(* IEC 61131-3 sources: cybercode_codesys_lib/src/basic/signal, 4 files *)

(* ---- FB_NumericChangeDetector.st ---- *)
FUNCTION_BLOCK FB_NumericChangeDetector
VAR_INPUT
    irValue : REAL;          // Входное числовое значение для мониторинга
END_VAR
VAR_OUTPUT
    qxChangeDetected : BOOL; // Импульс при обнаружении изменения значения
END_VAR
VAR
    _rPreviousValue : REAL := 0.0;    // Предыдущее значение для сравнения
    _xFirstCycle : BOOL := TRUE;      // Флаг первого цикла выполнения
    _rt_Change : R_TRIG;              // Триггер для генерации импульса
    _xValueChanged : BOOL := FALSE;   // Внутренний флаг изменения
END_VAR

// Пропускаем первый цикл для корректной инициализации
IF _xFirstCycle THEN
    _rPreviousValue := irValue;
    _xFirstCycle := FALSE;
    _xValueChanged := FALSE;
ELSE
    // Проверяем изменение значения
    IF _rPreviousValue <> irValue THEN
        _xValueChanged := TRUE;
        _rPreviousValue := irValue;
    ELSE
        _xValueChanged := FALSE;
    END_IF
END_IF

// Генерируем импульс при изменении через R_TRIG
_rt_Change(CLK := _xValueChanged);
qxChangeDetected := _rt_Change.Q;

(* Получение текущего отслеживаемого значения *)
METHOD GetCurrentValue : REAL
VAR_INPUT
END_VAR
    GetCurrentValue := irValue;
END_METHOD

(* Получение предыдущего значения *)
METHOD GetPreviousValue : REAL
VAR_INPUT
END_VAR
    GetPreviousValue := _rPreviousValue;
END_METHOD

(* Получение разности между текущим и предыдущим значением *)
METHOD GetValueDifference : REAL
VAR_INPUT
END_VAR
    GetValueDifference := irValue - _rPreviousValue;
END_METHOD

(* Проверка увеличения значения *)
METHOD IsValueIncreased : BOOL
VAR_INPUT
END_VAR
    IsValueIncreased := _xValueChanged AND (irValue > _rPreviousValue);
END_METHOD

(* Проверка уменьшения значения *)
METHOD IsValueDecreased : BOOL
VAR_INPUT
END_VAR
    IsValueDecreased := _xValueChanged AND (irValue < _rPreviousValue);
END_METHOD

(* Сброс детектора изменений *)
METHOD Reset
VAR_INPUT
END_VAR
    _rPreviousValue := irValue;
    _xFirstCycle := TRUE;
    _xValueChanged := FALSE;
    _rt_Change(CLK := FALSE);
END_METHOD

END_FUNCTION_BLOCK

(* ---- FB_SignalWithFeedback.st ---- *)
FUNCTION_BLOCK FB_SignalWithFeedback EXTENDS FB_BasicSignal
VAR_INPUT
    ixFeedback : BOOL;  	// Сигнал обратной связи
END_VAR
VAR_OUTPUT
END_VAR
VAR
	_inputSignalTrigger : FB_SignalWithTrigger; // Фиксация сигнала поступления команды
	_xWaitingFeedback : BOOL;	// Флаг ожидания сигнала обратной связи
    _xFeedbackReceived : BOOL;  // Флаг успешного получения обратной связи
END_VAR

    _inputSignalTrigger(ixSignal:= GetSignal());

    // Задание флага ожидания сигнала обртаной связи при получении сигнала команды
    IF _inputSignalTrigger.GetRtrig() AND NOT _xWaitingFeedback THEN
        _xWaitingFeedback := TRUE;
    END_IF

    // Задание флага получения обратной связи и ресет флага ожидания
    IF _xWaitingFeedback AND ixFeedback THEN
        _xFeedbackReceived := TRUE;
        ResetWaitingFeedback();
    END_IF

(* ---- FB_SignalWithRattling.st ---- *)
FUNCTION_BLOCK FB_SignalWithRattling EXTENDS FB_BasicSignal
VAR_INPUT
END_VAR
VAR_OUTPUT
END_VAR
VAR
    _ton_RattlingSignal : TON;
    _xOutSignal : BOOL;
END_VAR

_ton_RattlingSignal(IN:=GetSignal(), PT := T#100ms)

_outSignal := _ton_RattlingSignal.Q;

METHOD GetProcessedSignal : BOOL
    GetProcessedSignal := _outSignal;
END_METHOD

END_FUNCTION_BLOCK

(* ---- FB_SignalWithTrigger.st ---- *)
FUNCTION_BLOCK FB_SignalWithTrigger EXTENDS FB_BasicSignal
VAR_INPUT
END_VAR
VAR_OUTPUT
END_VAR
VAR
	_rt_xSignal : R_TRIG;
	_ft_xSignal : F_TRIG;
END_VAR

    _rt_xSignal(CLK:=GetSignal());
    _ft_xSignal(CLK:= GetSignal());

METHOD GetFtrig : BOOL
VAR_INPUT
END_VAR
    GetFtrig := _ft_xSignal.Q;
END_METHOD

METHOD GetRtrig : BOOL
VAR_INPUT
END_VAR
    GetRtrig := _rt_xSignal.Q;
END_METHOD

END_FUNCTION_BLOCK
